TYPE eInput :
STRUCT
	iState			: BOOL;
	iForceActive 	: BOOL;
	iForceInactive	: BOOL;
	cName			: STRING;
	cActiveState 	: BOOL := TRUE;
	oActive			: BOOL;
END_STRUCT
END_TYPE

(* stored: Version 1.1.0.1, ProductVersion 3.1.4022.11
   DUT eInput: Id {2b0f4537-518b-4738-adbe-fc0d7d271a6c} *)
